Fanuc KAREL source: kf00051.KL

-- PROVISIONAL review KL for V1013-1; original PC SHA256 402ce8af336e9b56d462412a82a15b7edae161b5aa6964d4c126a1553bbcbbe6
-- Incomplete behavior may be omitted. Consult companion uncertainty JSON. Do not deploy.
PROGRAM KF00051
%NOLOCKGROUP
VAR
  I : INTEGER
  J : INTEGER
  X : REAL
  Y : REAL
  B : BOOLEAN
  C : BOOLEAN
  TXT : STRING[80]
  TXT2 : STRING[80]
  STATUS : INTEGER
-- UNRESOLVED_DECL AI type=002010
-- UNRESOLVED_DECL BI type=002010
-- UNRESOLVED_DECL P type=000102
-- UNRESOLVED_DECL JP type=000199
-- UNRESOLVED_DECL PF type=000101
-- UNRESOLVED_DECL V1 type=000013
-- UNRESOLVED_DECL V2 type=000013
BEGIN
  -- UNRESOLVED_PC offsets 5-34; opcodes 2E,23,9F,9D,22,7A
  -- UNRESOLVED_PC offsets 39-58; opcodes 21,21,52,23
  -- UNRESOLVED_PC offsets 63-78; opcodes 45,2C,23
  -- UNRESOLVED_PC offsets 83-87; opcodes 7F
END KF00051
